SUBAPPLICATION Schneidwerk (* Subapplication Type *)
  (* Standard: 61499-2 *)
  (* Version 1.0, 2023-01-29, Franz *)
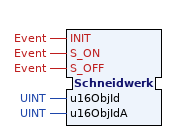
  EVENT_INPUT
    INIT;
    S_ON;
    S_OFF;
  END_EVENT
  VAR_INPUT
    u16ObjId : UINT;
    u16ObjIdA : UINT;
  END_VAR
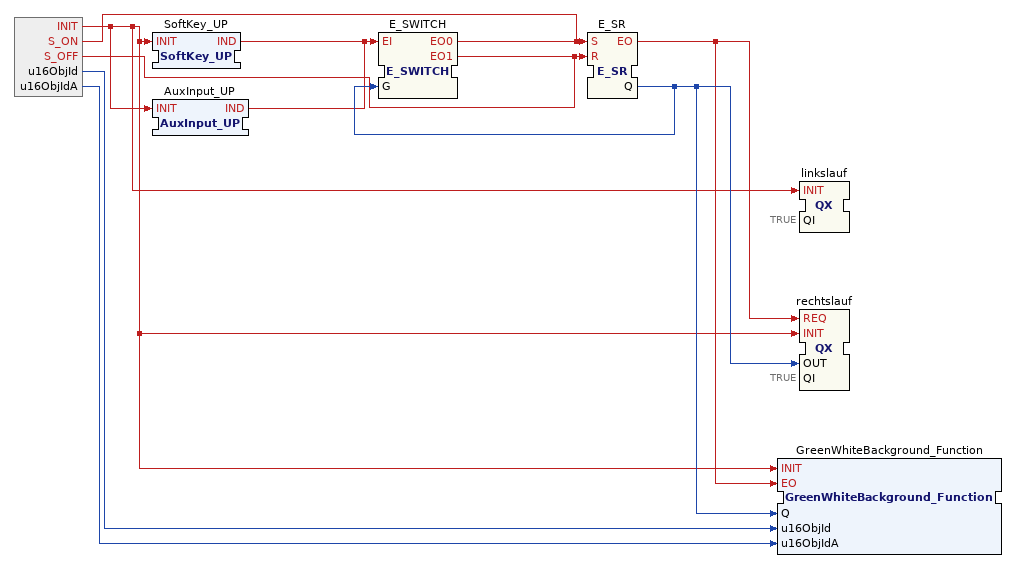
  (* Group __Group01: TODO: Schneidwerk linkslauf bei jedem 2. Start.  &#10; *)
  FBS
    rechtslauf : QX(QI := TRUE);
    E_SWITCH : E_SWITCH;
    E_SR : E_SR;
    linkslauf : QX(QI := TRUE);
  END_FBS
  SUBAPPS
    SoftKey_UP : SoftKey_UP;
    AuxInput_UP : AuxInput_UP;
    GreenWhiteBackground_Function : GreenWhiteBackground_Function;
  END_SUBAPPS
  EVENT_CONNECTIONS
    E_SR.EO TO rechtslauf.REQ;
    E_SWITCH.EO0 TO E_SR.S;
    E_SWITCH.EO1 TO E_SR.R;
    S_ON TO E_SR.S;
    S_OFF TO E_SR.R;
    INIT TO linkslauf.INIT;
    INIT TO rechtslauf.INIT;
    INIT TO SoftKey_UP.INIT;
    SoftKey_UP.IND TO E_SWITCH.EI;
    INIT TO AuxInput_UP.INIT;
    AuxInput_UP.IND TO E_SWITCH.EI;
    INIT TO GreenWhiteBackground_Function.INIT;
    E_SR.EO TO GreenWhiteBackground_Function.EO;
  END_CONNECTIONS
  DATA_CONNECTIONS
    E_SR.Q TO rechtslauf.OUT;
    E_SR.Q TO E_SWITCH.G;
    E_SR.Q TO GreenWhiteBackground_Function.Q;
    u16ObjId TO GreenWhiteBackground_Function.u16ObjId;
    u16ObjIdA TO GreenWhiteBackground_Function.u16ObjIdA;
  END_CONNECTIONS
END_SUBAPPLICATION
